Fanuc KAREL source: KA00139.KL

PROGRAM KA00139
%NOLOCKGROUP
VAR
  SRC: ARRAY[2] OF SHORT
  DST: XYZWPREXT
BEGIN
  SRC[1] = 2
  DST = SRC[1]
END KA00139
